SUBAPPLICATION Uebung_072b (* GBSD auf UT ausgeben *)
  (* Standard: 61499-2 *)
  (* Version 1.0, 2023-10-23, franz *)
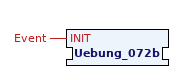
  EVENT_INPUT
    INIT;
  END_EVENT
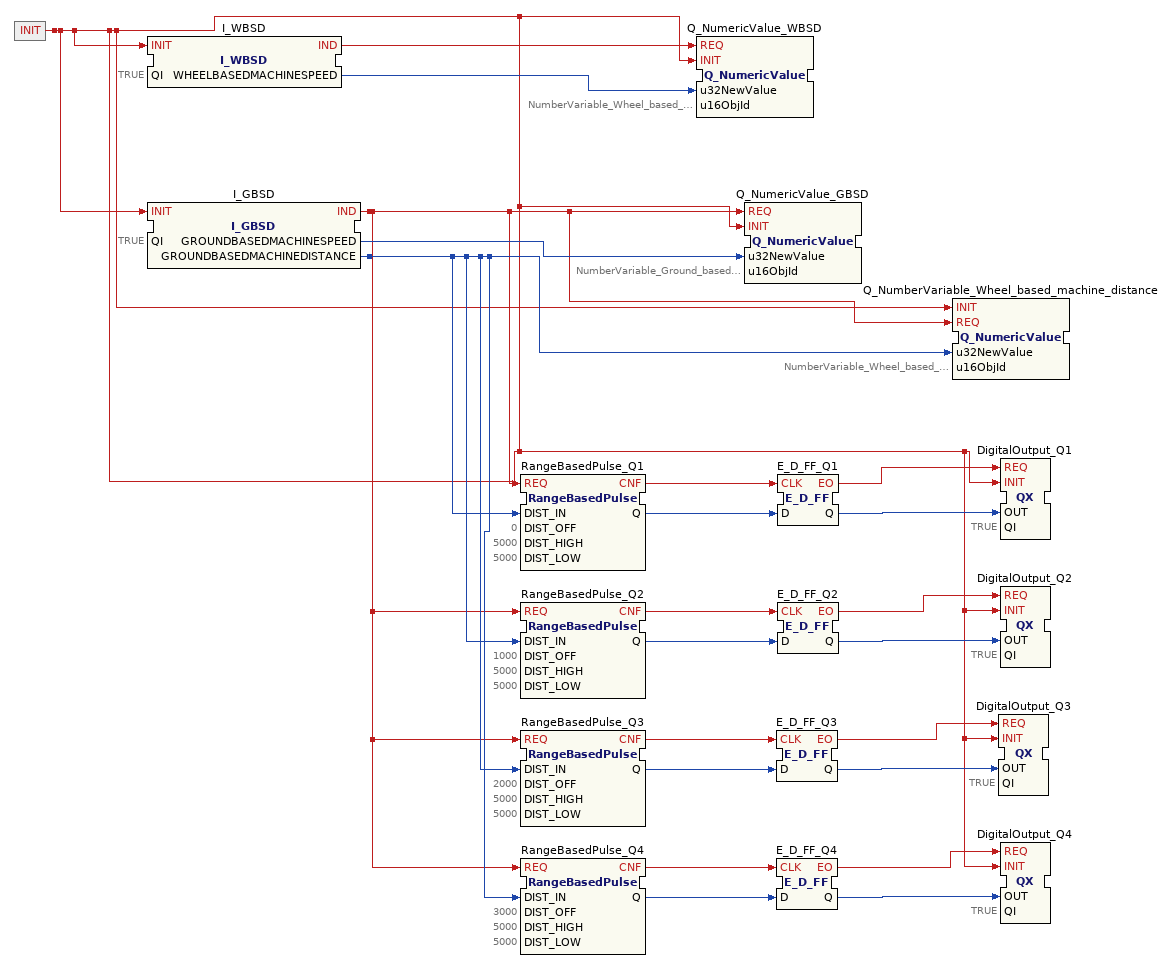
  FBS
    I_GBSD : I_GBSD(QI := TRUE);
    Q_NumericValue_GBSD : Q_NumericValue(u16ObjId := NumberVariable_Ground_based_machine_speed);
    I_WBSD : I_WBSD(QI := TRUE);
    Q_NumericValue_WBSD : Q_NumericValue(u16ObjId := NumberVariable_Wheel_based_machine_speed);
    Q_NumberVariable_Wheel_based_machine_distance : Q_NumericValue(u16ObjId := NumberVariable_Wheel_based_machine_distance);
    DigitalOutput_Q1 : QX(QI := TRUE);
    RangeBasedPulse_Q1 : signalprocessing::distance::RangeBasedPulse(DIST_OFF := 0, DIST_HIGH := 5000, DIST_LOW := 5000);
    E_D_FF_Q1 : E_D_FF;
    DigitalOutput_Q2 : QX(QI := TRUE);
    RangeBasedPulse_Q2 : signalprocessing::distance::RangeBasedPulse(DIST_OFF := 1000, DIST_HIGH := 5000, DIST_LOW := 5000);
    E_D_FF_Q2 : E_D_FF;
    DigitalOutput_Q3 : QX(QI := TRUE);
    RangeBasedPulse_Q3 : signalprocessing::distance::RangeBasedPulse(DIST_OFF := 2000, DIST_HIGH := 5000, DIST_LOW := 5000);
    E_D_FF_Q3 : E_D_FF;
    DigitalOutput_Q4 : QX(QI := TRUE);
    RangeBasedPulse_Q4 : signalprocessing::distance::RangeBasedPulse(DIST_OFF := 3000, DIST_HIGH := 5000, DIST_LOW := 5000);
    E_D_FF_Q4 : E_D_FF;
  END_FBS
  EVENT_CONNECTIONS
    INIT TO I_GBSD.INIT;
    I_GBSD.IND TO Q_NumericValue_GBSD.REQ;
    INIT TO I_WBSD.INIT;
    I_WBSD.IND TO Q_NumericValue_WBSD.REQ;
    E_D_FF_Q1.EO TO DigitalOutput_Q1.REQ;
    INIT TO DigitalOutput_Q1.INIT;
    INIT TO Q_NumericValue_WBSD.INIT;
    INIT TO Q_NumericValue_GBSD.INIT;
    INIT TO Q_NumberVariable_Wheel_based_machine_distance.INIT;
    I_GBSD.IND TO Q_NumberVariable_Wheel_based_machine_distance.REQ;
    E_D_FF_Q2.EO TO DigitalOutput_Q2.REQ;
    INIT TO DigitalOutput_Q2.INIT;
    E_D_FF_Q3.EO TO DigitalOutput_Q3.REQ;
    INIT TO DigitalOutput_Q3.INIT;
    E_D_FF_Q4.EO TO DigitalOutput_Q4.REQ;
    INIT TO DigitalOutput_Q4.INIT;
    I_GBSD.IND TO RangeBasedPulse_Q1.REQ;
    RangeBasedPulse_Q1.CNF TO E_D_FF_Q1.CLK;
    I_GBSD.IND TO RangeBasedPulse_Q2.REQ;
    RangeBasedPulse_Q2.CNF TO E_D_FF_Q2.CLK;
    I_GBSD.IND TO RangeBasedPulse_Q3.REQ;
    RangeBasedPulse_Q3.CNF TO E_D_FF_Q3.CLK;
    I_GBSD.IND TO RangeBasedPulse_Q4.REQ;
    RangeBasedPulse_Q4.CNF TO E_D_FF_Q4.CLK;
  END_CONNECTIONS
  DATA_CONNECTIONS
    I_GBSD.GROUNDBASEDMACHINESPEED TO Q_NumericValue_GBSD.u32NewValue;
    I_WBSD.WHEELBASEDMACHINESPEED TO Q_NumericValue_WBSD.u32NewValue;
    E_D_FF_Q1.Q TO DigitalOutput_Q1.OUT;
    I_GBSD.GROUNDBASEDMACHINEDISTANCE TO Q_NumberVariable_Wheel_based_machine_distance.u32NewValue;
    E_D_FF_Q2.Q TO DigitalOutput_Q2.OUT;
    E_D_FF_Q3.Q TO DigitalOutput_Q3.OUT;
    E_D_FF_Q4.Q TO DigitalOutput_Q4.OUT;
    I_GBSD.GROUNDBASEDMACHINEDISTANCE TO RangeBasedPulse_Q1.DIST_IN;
    RangeBasedPulse_Q1.Q TO E_D_FF_Q1.D;
    I_GBSD.GROUNDBASEDMACHINEDISTANCE TO RangeBasedPulse_Q2.DIST_IN;
    RangeBasedPulse_Q2.Q TO E_D_FF_Q2.D;
    I_GBSD.GROUNDBASEDMACHINEDISTANCE TO RangeBasedPulse_Q3.DIST_IN;
    RangeBasedPulse_Q3.Q TO E_D_FF_Q3.D;
    I_GBSD.GROUNDBASEDMACHINEDISTANCE TO RangeBasedPulse_Q4.DIST_IN;
    RangeBasedPulse_Q4.Q TO E_D_FF_Q4.D;
  END_CONNECTIONS
END_SUBAPPLICATION
